// TwinCAT 3 PLC project Elevator_L2
// ProgramVersion: 3.1.4023.0
// libraries:
//   Tc2_Standard, * (Beckhoff Automation GmbH)
//   Tc2_System, * (Beckhoff Automation GmbH)
//   Tc3_Module, * (Beckhoff Automation GmbH)
// project tree:
//   DUTs/ E_MotorStates.TcDUT, ST_Floor.TcDUT
//   / PlcTask.TcTTO
//   POUs/ FB_Motor.TcPOU, MAIN.TcPOU
// real-time tasks:
//   TASK PlcTask: cycle T#10ms, priority 20, ADS port 350

CONFIGURATION Elevator_L2
    RESOURCE PLC ON TwinCAT3
        TASK PlcTask(INTERVAL := T#10ms, PRIORITY := 20);
        PROGRAM MAIN WITH PlcTask : MAIN;
    END_RESOURCE
END_CONFIGURATION

// ---- DUTs/E_MotorStates.TcDUT
{attribute 'qualified_only'}
{attribute 'strict'}
TYPE E_MotorStates :
(
	stopped:=0,
	movingup,
	movingdown
);
END_TYPE

// ---- DUTs/ST_Floor.TcDUT
TYPE ST_Floor :
STRUCT
	High,
	Mid,
	Low:BOOL;
END_STRUCT
END_TYPE

// ---- POUs/MAIN.TcPOU
PROGRAM MAIN
VAR
	CallButtons:ARRAY[1..numFloor]OF BOOL;
	Floor:ARRAY[1..numFloor]OF ST_Floor;
	Elevator:FB_Motor;
	PrgState:UINT;
	current: INT;
	requested: INT;
	i: INT;
	Rise:ARRAY[1..numFloor] OF R_TRIG;
END_VAR
VAR CONSTANT
	numFloor:UINT:=6;
END_VAR

CASE	PrgState	OF
	0://stopped
		IF	current<requested	THEN
			PrgState:=20;//change state to moveing up
			Elevator.MoveUP();
		ELSIF current>requested	THEN
			PrgState:=30;//change state to moveing down
			Elevator.MoveDown();
		ELSE
			PrgState:=10;//poll for inputs
		END_IF
	10://poll input
		FOR	i:=1	TO	numFloor	DO
			IF	CallButtons[i]	THEN
				requested:=i;
				EXIT;
			END_IF
		END_FOR
		PrgState:=0;
	20://moveing up
		FOR i:=1	TO	numFloor	DO
			Rise[i](CLK:= Floor[i].Low,);
			IF	Rise[i].Q	THEN
				current:=current+1;
				IF	current=requested	THEN
					PrgState:=40;
				ELSE
					CONTINUE;
				END_IF
			ELSE
				CONTINUE;
			END_IF
		END_FOR
	30://moving down
		FOR i:=1	TO	numFloor	DO
			Rise[i](CLK:= Floor[i].High,);
			IF	Rise[i].Q	THEN
				current:=current-1;
				IF	current=requested	THEN
					PrgState:=40;
				ELSE
					CONTINUE;
				END_IF
			ELSE
				CONTINUE;
			END_IF
		END_FOR
	40://slowdown
		Elevator.SlowDown();
		FOR i:=1	TO	numFloor	DO
			IF	Floor[i].Mid	THEN
				Elevator.Stop();
				EXIT;
			END_IF
		END_FOR
		IF	elevator.IsStopped()	THEN
			PrgState:=0;
		END_IF
END_CASE

END_PROGRAM

// ---- POUs/FB_Motor.TcPOU
FUNCTION_BLOCK FB_Motor
VAR_INPUT
END_VAR
VAR_OUTPUT
END_VAR
VAR
	//movingup,
//	moving down
//stopped
// slow bit
	InternalState:E_MotorStates;
	slow:BOOL;
END_VAR

METHOD isSlow : BOOL
VAR_INPUT
END_VAR
isSlow:=slow;
END_METHOD

METHOD IsStopped : BOOL
VAR_INPUT
END_VAR
IsStopped:=FALSE;
IF	InternalState=E_MotorStates.stopped	THEN
	IsStopped:=TRUE;
END_IF
END_METHOD

METHOD MoveDown : BOOL
VAR_INPUT
END_VAR
InternalState:=E_MotorStates.movingdown;
slow:=false;
END_METHOD

METHOD MoveUP : BOOL
VAR_INPUT
END_VAR
InternalState:=E_MotorStates.movingup;
slow:=false;
END_METHOD

METHOD SlowDown : BOOL
VAR_INPUT
END_VAR
slow:=true;
END_METHOD

METHOD Stop : BOOL
VAR_INPUT
END_VAR
slow:=FALSE;
InternalState:=E_MotorStates.stopped;
END_METHOD

END_FUNCTION_BLOCK
